TYPE InfoDataAdsAddrStateBase_1916E49F :
STRUCT
END_STRUCT
END_TYPE

(* stored: Version 1.2.0.0, ProductVersion 3.1.4024.9
   DUT InfoDataAdsAddrStateBase_1916E49F: Id {3ab98fd7-ab94-4bcf-9c83-0b3d753c2d0c} *)
